TYPE ST_Example :
STRUCT
END_STRUCT
END_TYPE

(* stored: Version 1.1.0.1, ProductVersion 3.1.4024.11
   DUT ST_Example: Id {3a0c391e-5495-4eb8-87e4-0d06ae1e0ae9} *)
